// Mitsubishi GX Works2 project: 0630 조건 x10 누르면   PLC: Q02/Q02H

PROGRAM MAIN
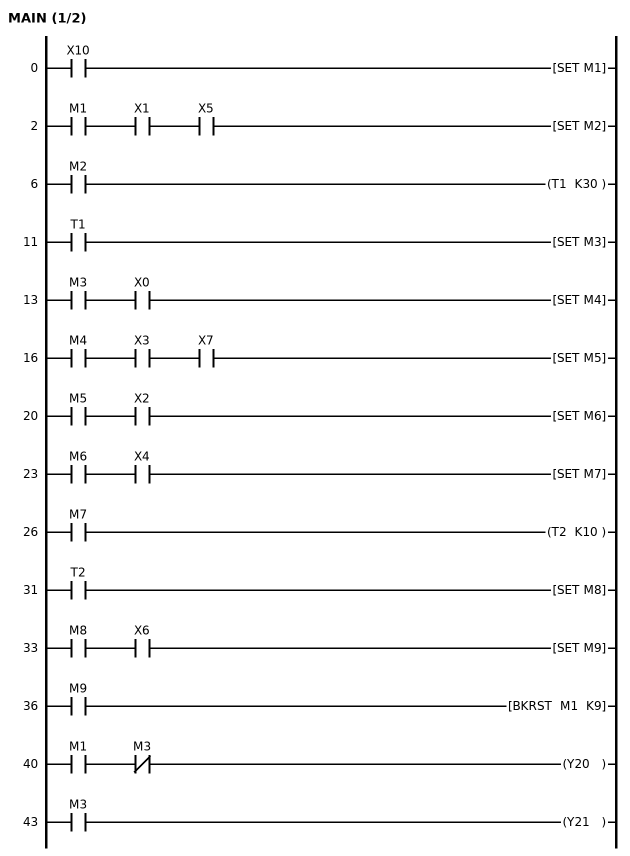
0     LD      X10
      SET     M1
2     LD      M1
      AND     X1
      AND     X5
      SET     M2
6     LD      M2
      OUT     T1 K30
11    LD      T1
      SET     M3
13    LD      M3
      AND     X0
      SET     M4
16    LD      M4
      AND     X3
      AND     X7
      SET     M5
20    LD      M5
      AND     X2
      SET     M6
23    LD      M6
      AND     X4
      SET     M7
26    LD      M7
      OUT     T2 K10
31    LD      T2
      SET     M8
33    LD      M8
      AND     X6
      SET     M9
36    LD      M9
      BKRST   M1 K9
40    LD      M1
      ANI     M3
      OUT     Y20
43    LD      M3
      OUT     Y21
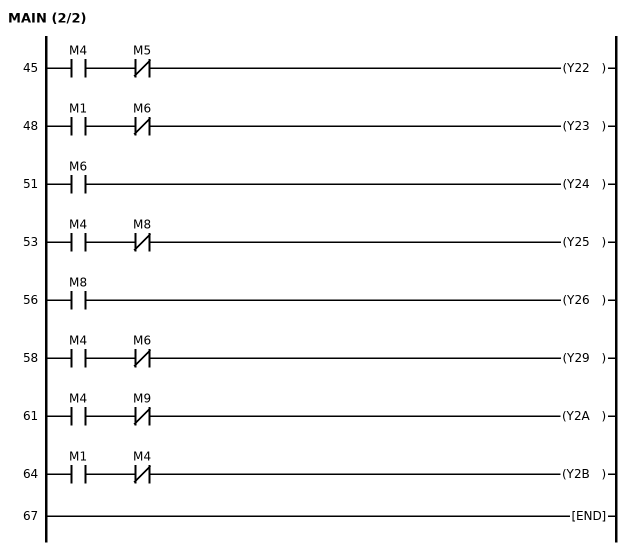
45    LD      M4
      ANI     M5
      OUT     Y22
48    LD      M1
      ANI     M6
      OUT     Y23
51    LD      M6
      OUT     Y24
53    LD      M4
      ANI     M8
      OUT     Y25
56    LD      M8
      OUT     Y26
58    LD      M4
      ANI     M6
      OUT     Y29
61    LD      M4
      ANI     M9
      OUT     Y2A
64    LD      M1
      ANI     M4
      OUT     Y2B
67    END
END_PROGRAM
